// LS Electric XG5000 project: 0122 시퀀스프로그램 양솔
// PLC LSPLC

PROGRAM NewProgram (task: 스캔 프로그램)

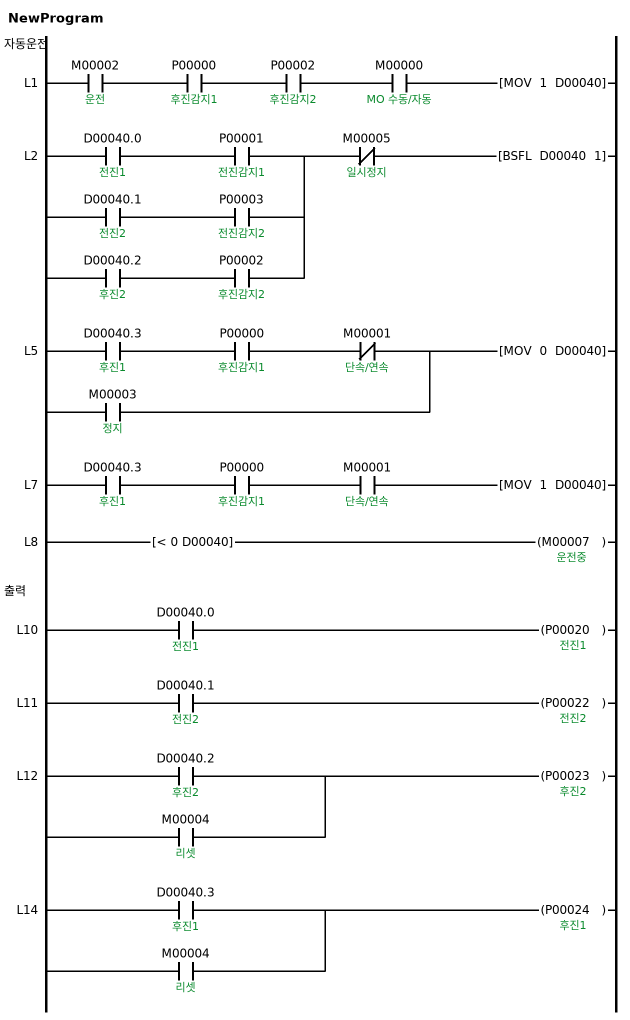
자동운전:
; L1
LOAD      M00002	// 운전
AND       P00000	// 후진감지1
AND       P00002	// 후진감지2
AND       M00000	// MO 수동/자동
MOV       1 D00040
; L2
LOAD      D00040.0	// 전진1
AND       P00001	// 전진감지1
LOAD      D00040.1	// 전진2
AND       P00003	// 전진감지2
OR LOAD
LOAD      D00040.2	// 후진2
AND       P00002	// 후진감지2
OR LOAD
AND NOT   M00005	// 일시정지
BSFL      D00040 1
; L5
LOAD      D00040.3	// 후진1
AND       P00000	// 후진감지1
AND NOT   M00001	// 단속/연속
OR        M00003	// 정지
MOV       0 D00040
; L7
LOAD      D00040.3	// 후진1
AND       P00000	// 후진감지1
AND       M00001	// 단속/연속
MOV       1 D00040
; L8
LOAD<     0 D00040
OUT       M00007	// 운전중
출력:
; L10
LOAD      D00040.0	// 전진1
OUT       P00020	// 전진1
; L11
LOAD      D00040.1	// 전진2
OUT       P00022	// 전진2
; L12
LOAD      D00040.2	// 후진2
OR        M00004	// 리셋
OUT       P00023	// 후진2
; L14
LOAD      D00040.3	// 후진1
OR        M00004	// 리셋
OUT       P00024	// 후진1

VARIABLES AND COMMENTS (devices not used above)
M00040	BIT	운전
M00041	BIT	NEXT
M00042	BIT	RESET